# B&R Automation Studio project Hartfiel_Tetris
Automation Studio 4.5.2.102; technology packages: Acp10Arnc0 5.6.2, mappView 5.6.3

## Configuration Config1

CPU X20CP1584, AutomationRuntime D4.52, Build 4.1.2, Vc V4.53.0, Safety 1.10

### Hardware
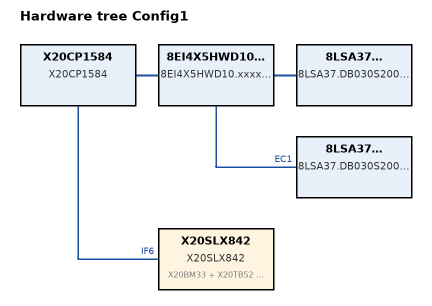
```
8EI4X5HWD10.xxxx-1 : 8EI4X5HWD10.xxxx-1 v2.3.0.2  [PLK1 -> X20CP1584.IF3 [Cable Type=PowerlinkCable, Length=10, Version=1.0.0.2]; EC1 -> 8LSA37.DB030S200-3a.EC; EC2 -> 8LSA37.DB030S200-3.EC; MT2 -> 8LSA37.DB030S200-3.MT]
  MotionTP = Acp10Arnc0
  BothEndSwitchesAreNormallyOpen_r1 = on
  QuickStopIsNormallyOpen_r1 = on
  BothEndSwitchesAreNormallyOpen_r2 = on
  QuickStopIsNormallyOpen_r2 = on
8LSA37.DB030S200-3 : 8LSA37.DB030S200-3 v1.0.5.34  [EC -> 8EI4X5HWD10.xxxx-1.EC2; MT -> 8EI4X5HWD10.xxxx-1.MT2]
8LSA37.DB030S200-3a : 8LSA37.DB030S200-3 v1.0.5.34  [EC -> 8EI4X5HWD10.xxxx-1.EC1; MT -> 8EI4X5HWD10.xxxx-1.MT1]
X20BM33 : X20BM33 v1.0.0.6  [X2X1 -> X20CP1584.IF6]
X20CP1584 : X20CP1584 v1.5.0.0
  Connector IF2:
    ActivateDevice = 1
  ConfigurationID = MpAxis_Setup_Config1
  Simulation = 1
  TimerDeviceType = EPLX2X
  TimerDevice = X20CP1584.IF3
  TaskClassIdleTime = 2000
  ActivateOpcUa = 1
  OpcUaInformationModels_PV_Version = 1
X20SLX842 : X20SLX842 v1.10.4.1  [SS1 -> X20TB52.SS; SS2 -> X20TB52a.SS; SL -> X20BM33.SL1]
  SafeProject = SafeLOGIC-1
X20TB52 : X20TB52 v1.0.0.1
X20TB52a : X20TB52 v1.0.0.1
```

### Acp10cfg.ncc - X20CP1584/Motion/Acp10cfg.ncc
```
NcConfiguration (Version=5.06.2, NcSwId=Acp10)
  ACP10CF1_typ:
    cnt_nettrc_rec_drive = 1500
    bufsize_trace_upload = 1200
    tc_nc_man_task = Cyclic #1
    glob_pv_as_ncobject = Yes
    ncsys_dl_broadcast = Yes
    ncsys_dl_acp_reset = Yes
    safemc_log_err_to_ax = Yes
    network_init:
      ncsw_init_execute = Yes
      automatic_execute = No
      node_nr_warning = Yes
      net_err_before_ncact = Yes
    nettrc:
      enter_parsecrec = Yes
      enter_ncaction = Yes
      save_ring_startidx = Yes
    cam_prof_download:
      cam_dat_dl_parallel = No
      tc_cam_dl_parallel = Task class for NC Manager task
    plk_if[0]:
      if_name = IF3
      tc_CycDat_PLCopen = Task class for NC Manager task
      mc_broadcast_extdat = No
```

### Acp10map.ncm - X20CP1584/Motion/Acp10map.ncm
```
NcMapping (NcSwId=Acp10)
  NcObject gAxis01 (ModuleId=8EI4X5HWD10.xxxx-1, Type=ncAXIS, Channel=1, AcoposSimulation=Off, InitParameter=gAxis01i, AcoposParameter=gAxis01a, Disabled=FALSE, ModuleDisabled=FALSE)
  NcObject gAxis02 (ModuleId=8EI4X5HWD10.xxxx-1, Type=ncAXIS, Channel=2, AcoposSimulation=Off, InitParameter=gAxis02i, AcoposParameter=gAxis02a, Disabled=FALSE, ModuleDisabled=FALSE)
  NcObject 8EI4X5HWD10.xxxx-1_ncV_AXIS1 (ModuleId=8EI4X5HWD10.xxxx-1, Type=ncV_AXIS, Channel=1, Disabled=TRUE, ModuleDisabled=FALSE)
  NcObject 8EI4X5HWD10.xxxx-1_ncV_AXIS2 (ModuleId=8EI4X5HWD10.xxxx-1, Type=ncV_AXIS, Channel=2, Disabled=TRUE, ModuleDisabled=FALSE)
```

### Config.mpaxisbasic - X20CP1584/Motion/Config.mpaxisbasic
```
Element gAxisBasic_0 (Type=mpaxisbasic)
Element gAxisBasic_1 (Type=mpaxisbasic)
```

## Logical view

Binary libraries used (declarations not repeated): operator, runtime, astime, AsIecCon, AsSafety, FileIO, DataObj, AsXml, standard, Acp10man 5.06.2, Acp10par 5.06.2, NcGlobal 5.06.2, Acp10_MC 5.06.2, brsystem, sys_lib, MpAxis 1.69.0, MpCom 5.06.2, MpBase 5.06.0

### Global.var - Global variables
```iecst
VAR
	gAxis01 : ACP10AXIS_typ;
	gAxis02 : ACP10AXIS_typ;
	TestButton1 : BOOL;
	TestButton2 : BOOL;
	TestButton3 : BOOL;
	TestButton4 : BOOL;
END_VAR
```


### Data object Logical/acp10etxen (Ett)

- acp10etxen.ett (not shown)

### Package Logical/gAxis02obj - gAxis02obj

### gAxis02i.ax
```
InitParameter (Version=5.6.2, NcSwId=Acp10)
  ACP10AXIS_typ:
    dig_in:
      level:
        reference = ncACTIV_HI
        pos_hw_end = ncACTIV_HI
        neg_hw_end = ncACTIV_HI
        trigger1 = ncACTIV_HI
        trigger2 = ncACTIV_HI
    encoder_if:
      parameter:
        count_dir = ncSTANDARD
        scaling:
          load:
            units = 1000
            rev_motor = 1
    limit:
      parameter:
        v_pos = 10000
        v_neg = 10000
        a1_pos = 50000
        a2_pos = 50000
        a1_neg = 50000
        a2_neg = 50000
        t_jolt = 0
        t_in_pos = 0
        pos_sw_end = 2000000000
        neg_sw_end = -2000000000
        ds_warning = 500
        ds_stop = 1000
        a_stop = 1.0e30
        dv_stop = 0
        dv_stop_mode = ncOFF
    controller:
      mode = ncPOSITION
      position:
        kv = 50
        tn = 0
        t_predict = 0.0004
        t_total = 0.0004
        p_max = 1.0e30
        i_max = 0
      speed:
        kv = 2.0
        tn = 0
        t_filter = 0.0
        isq_filter1:
          type = ncOFF
          a0 = 0.0
          a1 = 0.0
          b0 = 0.0
          b1 = 0.0
          b2 = 0.0
          c0_par_id = 0
          c1_par_id = 0
        isq_filter2:
          type = ncOFF
          a0 = 0.0
          a1 = 0.0
          b0 = 0.0
          b1 = 0.0
          b2 = 0.0
          c0_par_id = 0
          c1_par_id = 0
        isq_filter3:
          type = ncOFF
          a0 = 0.0
          a1 = 0.0
          b0 = 0.0
          b1 = 0.0
          b2 = 0.0
          c0_par_id = 0
          c1_par_id = 0
      uf:
        type = ncLINEAR + ncCORRECTION
        auto_config = ncMOTOR_PAR
        u0 = 0
        un = 0
        fn = 50.0
        k_f_slip = 0
      ff:
        mode = ncSTANDARD
        torque_load = 0.0
        torque_pos = 0.0
        torque_neg = 0.0
        kv_torque = 0.0
        inertia = 0.0
        t_filter_a = 0.0
      fb:
        mode = ncSTANDARD
        speed_mix_ratio = 0.0
        speed_kv = 2.0
      model:
        mass1:
          inertia = 0
          viscous_friction = 0
        mass2:
          inertia = 0
          viscous_friction = 0
          stiffness = 0
          damping = 0
    move:
      stop:
        parameter[0]:
          decel_ramp = ncA_LIMIT
          controller = ncON
        parameter[1]:
          decel_ramp = ncA_LIMIT
          controller = ncON
        parameter[2]:
          decel_ramp = ncA_LIMIT
          controller = ncON
        parameter[3]:
          decel_ramp = ncA_LIMIT
          controller = ncON
        quickstop:
          decel_ramp = ncA_LIMIT
          t_jolt = 0
        drive_error:
          decel_ramp = ncA_LIMIT
      homing:
        parameter:
          s = 0
          v_switch = 5000
          v_trigger = 500
          a = 50000
          mode = ncDIRECT
          edge_sw = ncPOSITIVE
          start_dir = ncPOSITIVE
          trigg_dir = ncPOSITIVE
          ref_pulse = ncOFF
          fix_dir = ncOFF
          tr_s_block = 0
          torque_lim = 0
          ds_block = 0
          ds_stop = 0
      basis:
        parameter:
          v_pos = 5000
          v_neg = 5000
          a1_pos = 50000
          a2_pos = 50000
          a1_neg = 50000
          a2_neg = 50000
    message:
      text:
        parameter:
          format = ncBREAK
          columns = 80
          data_modul = acp10etxen
```

- Visualisation Logical/mappView (not shown)

- MappView.lnk (binary file, 2350 bytes)
### Program Logical/Program (IEC)

#### Variables.var
```iecst
VAR
	test1calvar : BOOL;
	i : INT;
	yousure : BOOL;
END_VAR
```

#### Main.st
```iecst
PROGRAM _INIT
	(* Insert code here *)

END_PROGRAM

PROGRAM _CYCLIC
	test1calvar;
	TestButton1;
	TestButton2;
	TestButton3;
END_PROGRAM

PROGRAM _EXIT
	(* Insert code here *)

END_PROGRAM
```

Listed in the project but not available here: Logical/Global.typ, Logical/gAxis01obj
